// TIA Portal project "Clase1Sim" (V14)
// Simulación de la clase 1

(* hardware
DEVICE "S7-1200 station_1"  S7-1200 Station
   slot 0: "Rack_0"  S7-1200 Rack  Rack  V1.0
   slot 1: "Limon_PLC"  CPU 1214C DC/DC/DC  6ES7 214-1AG40-0XB0  V4.2
*)

// ===== PLC "Limon_PLC"  CPU 1214C DC/DC/DC =====

VAR_GLOBAL   // PLC tag table "Default tag table"
   ""start"" AT %I0.0 : Bool;
   ""stop"" AT %I0.1 : Bool;
   ""L1"" AT %Q0.0 : Bool;
   ""L2"" AT %Q0.1 : Bool;
END_VAR